RoboDK station: A_B_C_frames.rdk

Station A (saved by RoboDK 5.8.0). Poses are relative to the parent item; angles as X-Y-Z fixed-axis rotations.
  - frame B at (30, 50, 30) mm, rotated rx 30 ry 0 rz 0 deg
    - frame C at (0, 100, 60) mm, rotated rx 90 ry -30 rz 90 deg
